// TIA Portal V17 export
// export: Created 2025-03-05T08:03:00.2001919Z, ExportSetting WithDefaults, DisplayName Totally Integrated Automation Portal, DisplayVersion V17 Update 8, DisplayName TIA Portal Openness, DisplayVersion V17 Update 8, DisplayName TIA Portal Version Control Interface, DisplayVersion V17, DisplayName SINAMICS Startdrive Advanced, DisplayVersion V17 SP2, DisplayName SINAMICS Startdrive G110M, G120, G120C, G120D, G120P, G115D, DisplayVersion V17 SP2, DisplayName SINAMICS Startdrive G130, G150, S120, S150, SINAMICS MV, S210, DisplayVersion V17 SP2, DisplayName STEP 7 Professional, DisplayVersion V17 Update 8, DisplayName SINUMERIK ONE STEP 7 Toolbox, DisplayVersion V17 Update 12, DisplayName SINUMERIK 840D sl STEP 7 Toolbox, DisplayVersion V17 Update 12, DisplayName STEP 7 Safety, DisplayVersion V17 Update 6, DisplayName WinCC Advanced, DisplayVersion V17 Update 8
DATA_BLOCK "DB16702_OPC_UA_MASTER_POWDER"   // DB16702
{ S7_Optimized_Access := 'TRUE' }
VERSION : 0.1
// stored: AutoNumber false, DBAccessibleFromOPCUA true, DBAccessibleFromWebserver true, IsOnlyStoredInLoadMemory false, IsRetainMemResEnabled false, IsWriteProtectedInAS false, MemoryReserve 100
   VAR
      GENERAL { ExternalWritable := 'False'} : Struct
         LINE_ID { ExternalWritable := 'False'} : Int;   // GENERAL INFORMATION: PRODUCTION LINE IDENTIFICATION
         MACHINE_ID { ExternalWritable := 'False'} : Int;   // GENERAL INFORMATION: PRODUCTION MACHINE IDENTIFICATION
         PLC_ID { ExternalWritable := 'False'} : Int;   // GENERAL INFORMATION: PRODUCTION PLC IDENTIFICATION (POWDER PLC = 1 / MACHINE PLC = 2)
      END_STRUCT;
      UNIT_01 { ExternalWritable := 'False'} : Struct
         HOPPER_1 { ExternalWritable := 'False'} : "HOPPER";
         HOPPER_2 { ExternalWritable := 'False'} : "HOPPER";
         FEEDER_1 { ExternalWritable := 'False'} : Struct
            LINE_1 { ExternalWritable := 'False'} : "POWDER_FEEDER_LINE";
            LINE_2 { ExternalWritable := 'False'} : "POWDER_FEEDER_LINE";
            WEIGHT { ExternalWritable := 'False'} : Real;
         END_STRUCT;
         FEEDER_NOZZLE_LINE { ExternalWritable := 'False'} : Struct
            COMBINER_POWDER_FLOW { ExternalWritable := 'False'} : Array[1..20] of "MEDICOAT_TIME_STAMP";   // UNIT 01 COMBINER POWDER FLOW VALUE (¿?¿?¿?¿?¿)
            NOZZLE_POWDER_FLOW { ExternalWritable := 'False'} : Array[1..20] of "MEDICOAT_TIME_STAMP";   // UNIT 01 PROCESS POWDER FLOW VALUE (¿?¿?¿?¿?¿)
         END_STRUCT;
      END_STRUCT;
      UNIT_02 { ExternalWritable := 'False'} : Struct
         HOPPER_1 { ExternalWritable := 'False'} : "HOPPER";
         HOPPER_2 { ExternalWritable := 'False'} : "HOPPER";
         HOPPER_3 { ExternalWritable := 'False'} : "HOPPER";
         FEEDER_1 { ExternalWritable := 'False'} : Struct
            LINE_1 { ExternalWritable := 'False'} : "POWDER_FEEDER_LINE";
            LINE_2 { ExternalWritable := 'False'} : "POWDER_FEEDER_LINE";
            WEIGHT { ExternalWritable := 'False'} : Real;
         END_STRUCT;
         FEEDER_2 { ExternalWritable := 'False'} : Struct
            LINE_1 { ExternalWritable := 'False'} : "POWDER_FEEDER_LINE";
            WEIGHT { ExternalWritable := 'False'} : Real;
         END_STRUCT;
         FEEDER_NOZZLE_LINE { ExternalWritable := 'False'} : Struct
            COMBINER_POWDER_FLOW { ExternalWritable := 'False'} : Array[1..20] of "MEDICOAT_TIME_STAMP";   // UNIT 02 COMBINER POWDER FLOW VALUE (¿?¿?¿?¿?¿)
            NOZZLE_POWDER_FLOW { ExternalWritable := 'False'} : Array[1..20] of "MEDICOAT_TIME_STAMP";   // UNIT 02 PROCESS POWDER FLOW VALUE (¿?¿?¿?¿?¿)
         END_STRUCT;
      END_STRUCT;
   END_VAR
BEGIN
END_DATA_BLOCK
